FUNCTION_BLOCK FB_TestB IMPLEMENTS ITF_MyTest
VAR_INPUT
END_VAR
VAR_OUTPUT
END_VAR
VAR
END_VAR

{warning 'Agregar implementación de método'}
METHOD METH1 : BOOL
END_METHOD

{warning 'Agregar implementación de método'}
METHOD METH2 : STRING
METH2 := 'FB_TestB';
END_METHOD

{warning 'Agregar implementación de método'}
METHOD METH3 : REAL
METH3 := 8.69;
END_METHOD

{warning 'Agregar implementación de propiedad'}
PROPERTY Prop1 : BOOL
GET
END_GET
SET
END_SET
END_PROPERTY

{warning 'Agregar implementación de propiedad'}
PROPERTY Prop2 : REAL
GET
END_GET
SET
END_SET
END_PROPERTY

{warning 'Agregar implementación de propiedad'}
PROPERTY Prop3 : STRING
GET
END_GET
SET
END_SET
END_PROPERTY

END_FUNCTION_BLOCK

(* stored: Version 1.1.0.1, ProductVersion 3.1.4024.12
   POU FB_TestB: Id {882b5e9a-33e2-4768-83aa-8f6371e5a21c}, SpecialFunc None
   Method METH1: Id {ed41c89c-c578-430c-8b2e-b598b1b34220}
   Method METH2: Id {a6c0b124-d593-4e40-aeb3-0bd2657d2f5a}
   Method METH3: Id {c18dd97a-15f0-4acc-9f48-576e6c03961b}
   Property Prop1: Id {52e2ace9-0c0a-43b2-8255-ec9784494114}
   Get Get: Id {718b9081-e379-458a-816c-266e8869054f}
   Set Set: Id {b5c20016-8cff-4f2d-abe6-ad528a891427}
   Property Prop2: Id {25bdf9ff-793c-4219-b73d-f28a55868f0d}
   Get Get: Id {8452f15e-cf26-4fa2-a23a-121a1d8ad3f6}
   Set Set: Id {4d92c7c1-f73d-4f12-b027-e475a675a9ed}
   Property Prop3: Id {4b306c44-e995-4afa-b371-d3a92156014c}
   Get Get: Id {6219a614-caee-4bce-8ca3-e221cb3141e4}
   Set Set: Id {2db227c2-47bc-41e8-886c-d63978baec61} *)
